FUNCTION_BLOCK FB_Child EXTENDS FB_Parent
VAR_INPUT
END_VAR
VAR_OUTPUT
END_VAR
VAR
	m_child_data : ARRAY [0..1023] OF REAL;
END_VAR

METHOD FB_init : BOOL
VAR_INPUT
	bInitRetains : BOOL; // if TRUE, the retain variables are initialized (warm start / cold start)
	bInCopyCode : BOOL;  // if TRUE, the instance afterwards gets moved into the copy code (online change)
END_VAR
SUPER^.ref_child REF= THIS^;
END_METHOD

END_FUNCTION_BLOCK

(* stored: Version 1.1.0.1, ProductVersion 3.1.4024.12
   POU FB_Child: Id {cda601de-aae1-4afb-98c9-56c3d3ddc641}, SpecialFunc None
   Method FB_init: Id {120ddc91-1804-4e8d-86a5-3db744e6c221} *)
